// Mitsubishi GX Works2 project: PLC_Group_33   PLC: FX3G

// global labels: Global1
VAR_GLOBAL
  EmergeStop AT X005 : BOOL;
  PrepStart AT X001 : BOOL;
  CoolStart AT X002 : BOOL;
  TempSensor AT X003 : BOOL;
  AnalogIn1 AT D8280 : INT;
  AnalogOut AT D8282 : INT;
  DayCoil AT Y007 : BOOL;
  PrepCoil AT Y000 : BOOL;
  CoolCoil AT Y002 : BOOL;
  MixCoil1 AT Y005 : BOOL;
  MixCoil2 AT Y006 : BOOL;
  DayActive AT M0 : BOOL;
  DayEnd AT M1 : BOOL;
  TypeRegular AT M10 : BOOL;
  TypePremium AT M11 : BOOL;
  StockFail AT M20 : BOOL;
  PrepActive AT M30 : BOOL;
  PrepDone AT M31 : BOOL;
  CoolActive AT M40 : BOOL;
  CoolDone AT M41 : BOOL;
  MixActive AT M50 : BOOL;
  MixDone AT M51 : BOOL;
  BlinkHelper AT M60 : BOOL;
  ResetAll AT M70 : BOOL;
  PrepTimerC AT TC0 : BOOL;
  PrepTimerS AT TS0 : BOOL;
END_VAR
VAR_GLOBAL CONSTANT
  PrepTimerCVal : INT := K50;
END_VAR
VAR_GLOBAL
  CoolTimerC AT TC1 : BOOL;
  CoolTimerS AT TS1 : BOOL;
END_VAR
VAR_GLOBAL CONSTANT
  CoolTimerVal : INT := K80;
END_VAR
VAR_GLOBAL
  MixTimerC AT TC2 : BOOL;
  MixTimerS AT TS2 : BOOL;
END_VAR
VAR_GLOBAL CONSTANT
  MixTimerReg : INT := K30;
  MixTimePrem : INT := K50;
END_VAR
VAR_GLOBAL
  BlinkTC1 AT TC3 : BOOL;
  BlinkTS1 AT TS3 : BOOL;
  BlinkTC2 AT TC4 : BOOL;
  BlinkTS2 AT TS4 : BOOL;
END_VAR
VAR_GLOBAL CONSTANT
  BlinkVal : INT := K5;
END_VAR
VAR_GLOBAL
  RaspSt AT D1100 : INT;
  LemonSt AT D1102 : INT;
  StabSt AT D1104 : INT;
  GummySt AT D1106 : INT;
  RaspStock AT D1110 : INT;
  LemonStock AT D1112 : INT;
  StabStock AT D1114 : INT;
  GummyStock AT D1116 : INT;
  NeededRasp AT D1120 : INT;
  NeededLemon AT D1122 : INT;
  NeededStab AT D1124 : INT;
  NeededGummy AT D1126 : INT;
END_VAR
VAR_GLOBAL CONSTANT
  RegRasp : INT := K280;
  RegLemon : INT := K455;
  RegStab : INT := K105;
  RegGummy : INT := K28;
  PremRasp : INT := K385;
  PremLemon : INT := K665;
  PremStab : INT := K210;
  PremGummy : INT := K70;
END_VAR
VAR_GLOBAL
  CoolRasp AT D1130 : INT;
  CoolLemon AT D1132 : INT;
  MixTank AT D1134 : INT;
  BoxCount AT D1140 : INT;
  DayStart AT X007 : BOOL;
  AnalogSample AT D1150 : INT;
  RaspLow AT M80 : BOOL;
  LemonLow AT M81 : BOOL;
  StabLow AT M82 : BOOL;
  GummyLow AT M83 : BOOL;
  MixTimerVal AT D200 : INT;
END_VAR
VAR_GLOBAL CONSTANT
  CoolRaspReg : INT := K350;
  CoolLemonReg : INT := K490;
  CoolRaspPrem : INT := K560;
  CoolLemonPrem : INT := K700;
END_VAR

// task Task_01 (event TRUE, interval 0, priority 31): POU_01

PROGRAM POU_01
(* structured ladder/FBD written out as ST: instructions are called as NAME(EN, inputs, outputs); _pN, _eN, _tN stand for wires *)
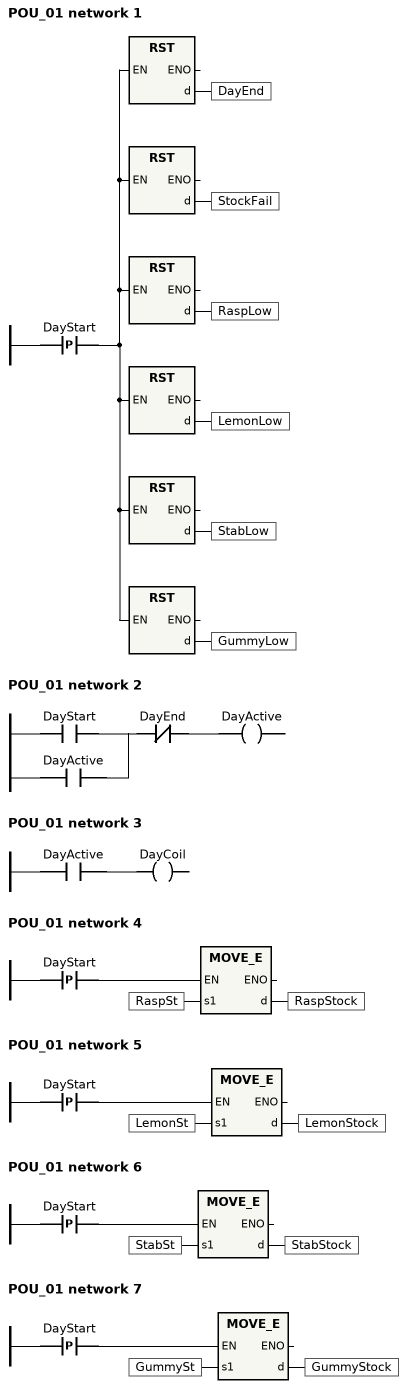
(* network 1 *)
_p1 := LDP(TRUE, DayStart);
RST(_p1, DayEnd);
RST(_p1, StockFail);
RST(_p1, RaspLow);
RST(_p1, LemonLow);
RST(_p1, StabLow);
RST(_p1, GummyLow);
(* network 2 *)
DayActive := (DayStart OR DayActive) AND NOT DayEnd;
(* network 3 *)
DayCoil := DayActive;
(* network 4 *)
MOVE_E(LDP(TRUE, DayStart), RaspSt, RaspStock);
(* network 5 *)
MOVE_E(LDP(TRUE, DayStart), LemonSt, LemonStock);
(* network 6 *)
MOVE_E(LDP(TRUE, DayStart), StabSt, StabStock);
(* network 7 *)
MOVE_E(LDP(TRUE, DayStart), GummySt, GummyStock);
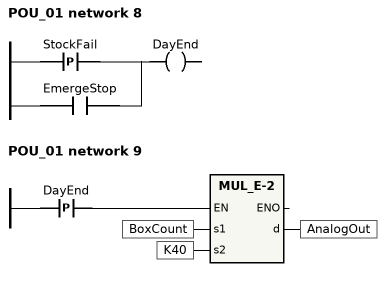
(* network 8 *)
DayEnd := LDP(TRUE, StockFail) OR EmergeStop;
(* network 9 *)
MUL_E(LDP(TRUE, DayEnd), BoxCount, K40, AnalogOut);
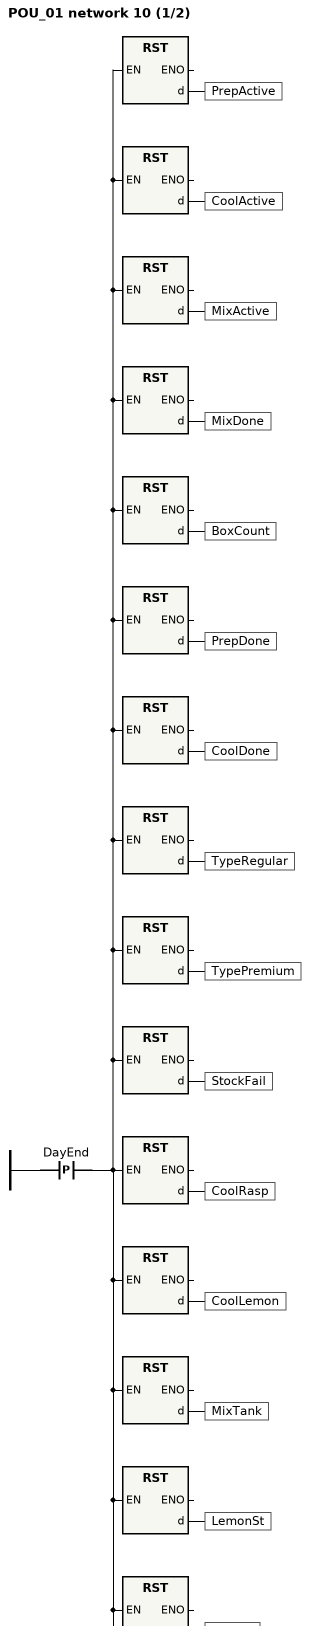
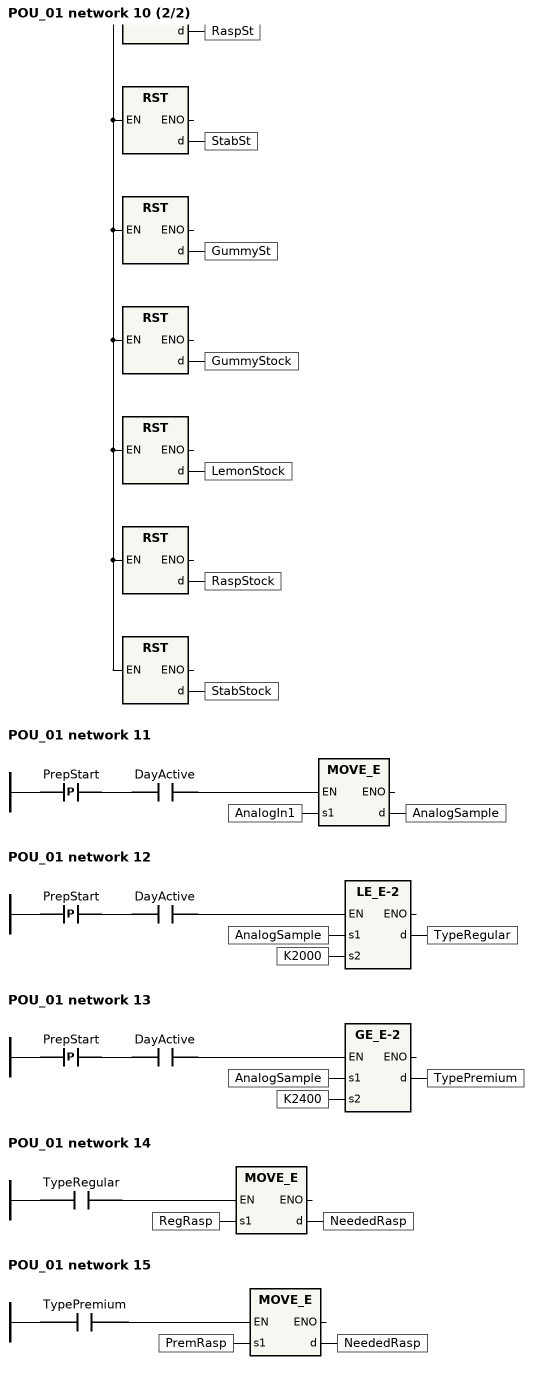
(* network 10 *)
_p1 := LDP(TRUE, DayEnd);
RST(_p1, PrepActive);
RST(_p1, CoolActive);
RST(_p1, MixActive);
RST(_p1, MixDone);
RST(_p1, BoxCount);
RST(_p1, PrepDone);
RST(_p1, CoolDone);
RST(_p1, TypeRegular);
RST(_p1, TypePremium);
RST(_p1, StockFail);
RST(_p1, CoolRasp);
RST(_p1, CoolLemon);
RST(_p1, MixTank);
RST(_p1, LemonSt);
RST(_p1, RaspSt);
RST(_p1, StabSt);
RST(_p1, GummySt);
RST(_p1, GummyStock);
RST(_p1, LemonStock);
RST(_p1, RaspStock);
RST(_p1, StabStock);
(* network 11 *)
MOVE_E(LDP(TRUE, PrepStart) AND DayActive, AnalogIn1, AnalogSample);
(* network 12 *)
LE_E(LDP(TRUE, PrepStart) AND DayActive, AnalogSample, K2000, TypeRegular);
(* network 13 *)
GE_E(LDP(TRUE, PrepStart) AND DayActive, AnalogSample, K2400, TypePremium);
(* network 14 *)
MOVE_E(TypeRegular, RegRasp, NeededRasp);
(* network 15 *)
MOVE_E(TypePremium, PremRasp, NeededRasp);
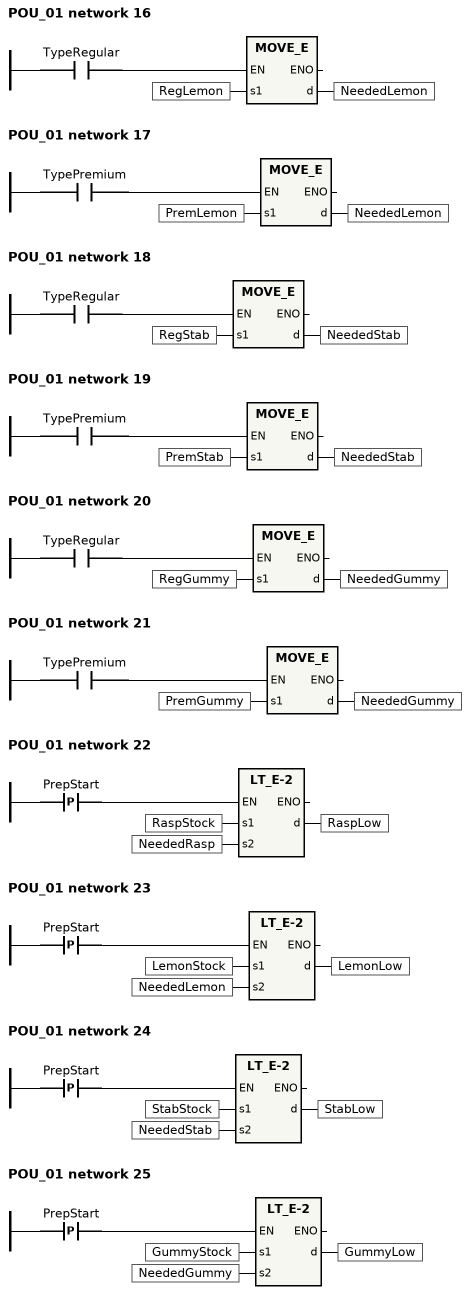
(* network 16 *)
MOVE_E(TypeRegular, RegLemon, NeededLemon);
(* network 17 *)
MOVE_E(TypePremium, PremLemon, NeededLemon);
(* network 18 *)
MOVE_E(TypeRegular, RegStab, NeededStab);
(* network 19 *)
MOVE_E(TypePremium, PremStab, NeededStab);
(* network 20 *)
MOVE_E(TypeRegular, RegGummy, NeededGummy);
(* network 21 *)
MOVE_E(TypePremium, PremGummy, NeededGummy);
(* network 22 *)
LT_E(LDP(TRUE, PrepStart), RaspStock, NeededRasp, RaspLow);
(* network 23 *)
LT_E(LDP(TRUE, PrepStart), LemonStock, NeededLemon, LemonLow);
(* network 24 *)
LT_E(LDP(TRUE, PrepStart), StabStock, NeededStab, StabLow);
(* network 25 *)
LT_E(LDP(TRUE, PrepStart), GummyStock, NeededGummy, GummyLow);
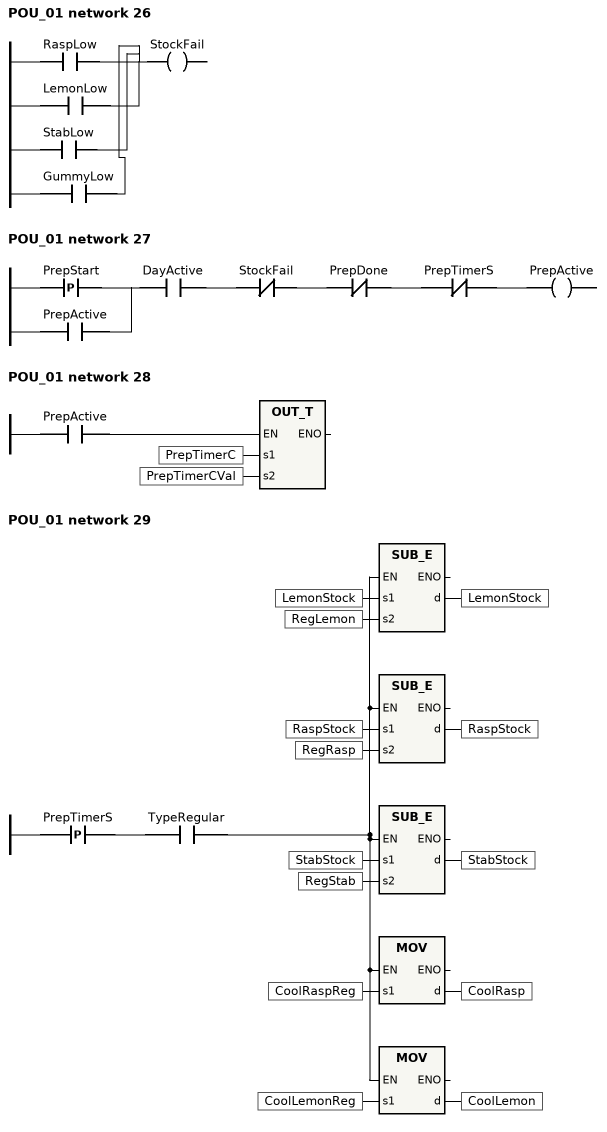
(* network 26 *)
StockFail := RaspLow OR LemonLow OR StabLow OR GummyLow;
(* network 27 *)
PrepActive := ((((LDP(TRUE, PrepStart) OR PrepActive) AND DayActive) AND NOT StockFail) AND NOT PrepDone) AND NOT PrepTimerS;
(* network 28 *)
OUT_T(PrepActive, PrepTimerC, PrepTimerCVal);
(* network 29 *)
_p1 := LDP(TRUE, PrepTimerS) AND TypeRegular;
SUB_E(_p1, LemonStock, RegLemon, LemonStock);
SUB_E(_p1, RaspStock, RegRasp, RaspStock);
SUB_E(_p1, StabStock, RegStab, StabStock);
MOV(_p1, CoolRaspReg, CoolRasp);
MOV(_p1, CoolLemonReg, CoolLemon);
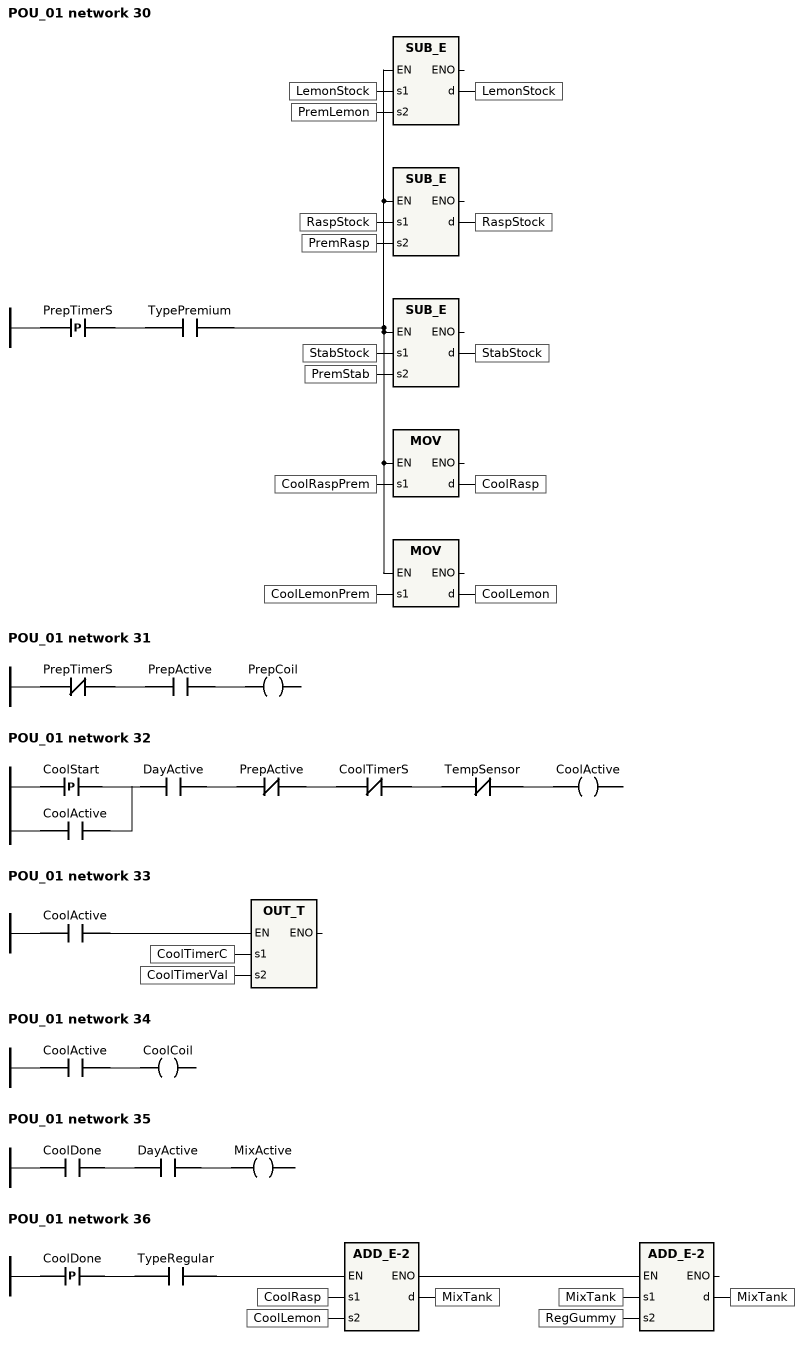
(* network 30 *)
_p1 := LDP(TRUE, PrepTimerS) AND TypePremium;
SUB_E(_p1, LemonStock, PremLemon, LemonStock);
SUB_E(_p1, RaspStock, PremRasp, RaspStock);
SUB_E(_p1, StabStock, PremStab, StabStock);
MOV(_p1, CoolRaspPrem, CoolRasp);
MOV(_p1, CoolLemonPrem, CoolLemon);
(* network 31 *)
PrepCoil := NOT PrepTimerS AND PrepActive;
(* network 32 *)
CoolActive := ((((LDP(TRUE, CoolStart) OR CoolActive) AND DayActive) AND NOT PrepActive) AND NOT CoolTimerS) AND NOT TempSensor;
(* network 33 *)
OUT_T(CoolActive, CoolTimerC, CoolTimerVal);
(* network 34 *)
CoolCoil := CoolActive;
(* network 35 *)
MixActive := CoolDone AND DayActive;
(* network 36 *)
_e1 := ADD_E(LDP(TRUE, CoolDone) AND TypeRegular, CoolRasp, CoolLemon, MixTank);
ADD_E(_e1, MixTank, RegGummy, MixTank);
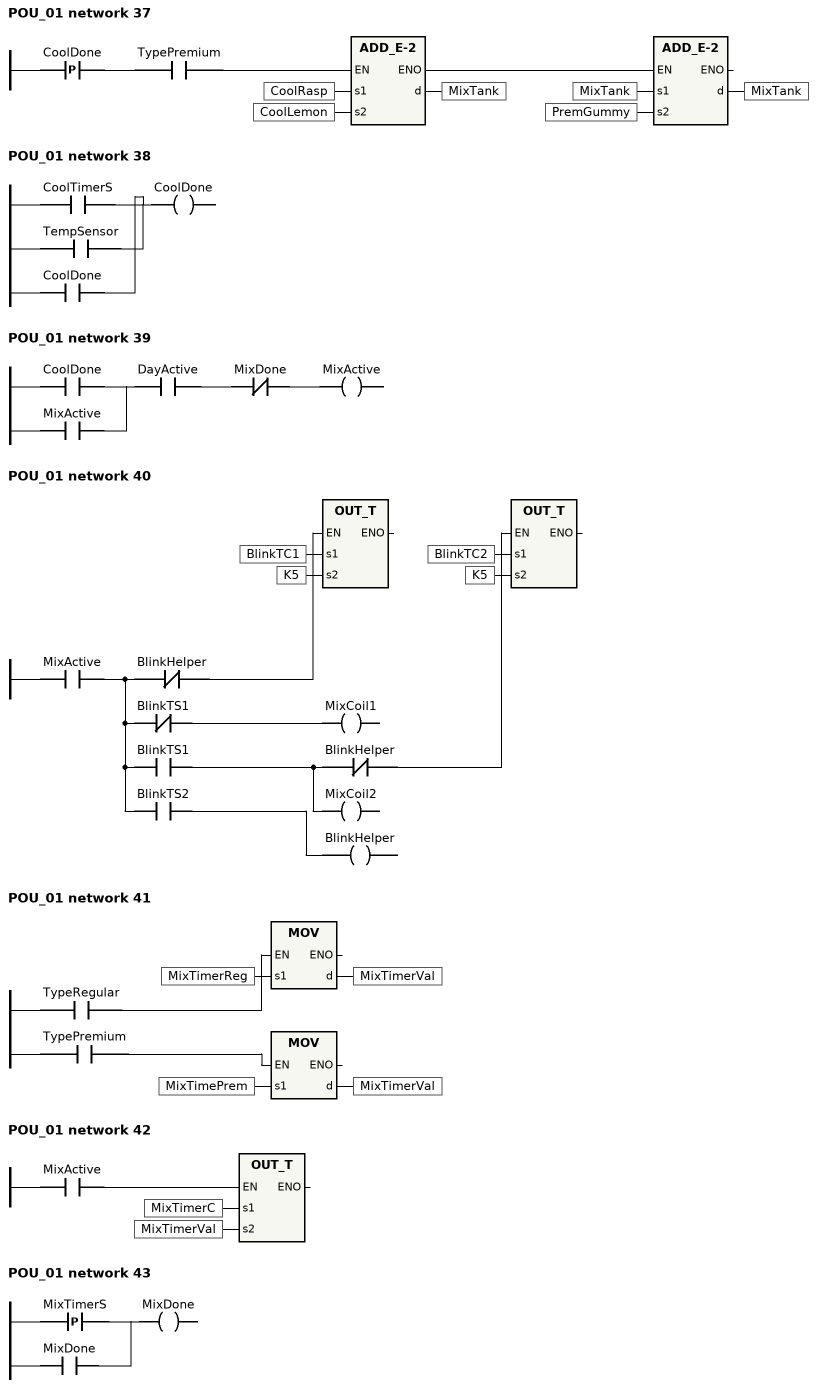
(* network 37 *)
_e1 := ADD_E(LDP(TRUE, CoolDone) AND TypePremium, CoolRasp, CoolLemon, MixTank);
ADD_E(_e1, MixTank, PremGummy, MixTank);
(* network 38 *)
CoolDone := CoolTimerS OR TempSensor OR CoolDone;
(* network 39 *)
MixActive := ((CoolDone OR MixActive) AND DayActive) AND NOT MixDone;
(* network 40 *)
OUT_T(MixActive AND NOT BlinkHelper, BlinkTC1, K5);
MixCoil1 := MixActive AND NOT BlinkTS1;
_p1 := MixActive AND BlinkTS1;
OUT_T(_p1 AND NOT BlinkHelper, BlinkTC2, K5);
MixCoil2 := _p1;
BlinkHelper := MixActive AND BlinkTS2;
(* network 41 *)
MOV(TypeRegular, MixTimerReg, MixTimerVal);
MOV(TypePremium, MixTimePrem, MixTimerVal);
(* network 42 *)
OUT_T(MixActive, MixTimerC, MixTimerVal);
(* network 43 *)
MixDone := LDP(TRUE, MixTimerS) OR MixDone;
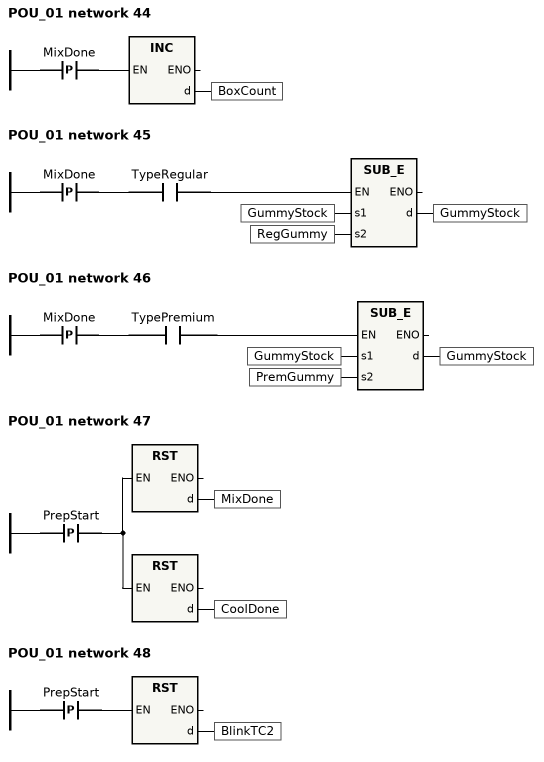
(* network 44 *)
INC(LDP(TRUE, MixDone), BoxCount);
(* network 45 *)
SUB_E(LDP(TRUE, MixDone) AND TypeRegular, GummyStock, RegGummy, GummyStock);
(* network 46 *)
SUB_E(LDP(TRUE, MixDone) AND TypePremium, GummyStock, PremGummy, GummyStock);
(* network 47 *)
_p1 := LDP(TRUE, PrepStart);
RST(_p1, MixDone);
RST(_p1, CoolDone);
(* network 48 *)
RST(LDP(TRUE, PrepStart), BlinkTC2);
END_PROGRAM
